INTERFACE ITF_Logger

END_INTERFACE

(* stored: Version 1.1.0.1
   Itf ITF_Logger: Id {dde1500f-ba43-0973-2072-39e8d4239f74} *)
